FUNCTION_BLOCK FB_Fixture222 EXTENDS FB_UniversalFixture
VAR_INPUT
END_VAR
VAR_OUTPUT
END_VAR
VAR
	(*
		Add fixture sensors and actuators
	*)
END_VAR

SUPER^();

(*
	Add FB instances
*)

METHOD PROTECTED MS_Close
VAR_INPUT
END_VAR
eFixtureState := UNIVERSAL_FIXTURE_CLOSE_DONE;
END_METHOD

METHOD PROTECTED MS_Open
VAR_INPUT
END_VAR
eFixtureState := UNIVERSAL_FIXTURE_OPEN_DONE;
END_METHOD

METHOD PROTECTED MS_ReadyInitialized
VAR_INPUT
END_VAR
eFixtureState := UNIVERSAL_FIXTURE_IDLE;
END_METHOD

METHOD PROTECTED MS_Reset
VAR_INPUT
END_VAR
eFixtureState := UNIVERSAL_FIXTURE_RESET_DONE;
END_METHOD

PROPERTY SocketOpen : REFERENCE TO BOOL
GET
SocketOpen REF= bSocketOpen;
END_GET
END_PROPERTY

END_FUNCTION_BLOCK

(* stored: Version 1.1.0.1, ProductVersion 3.1.4024.9
   POU FB_Fixture222: Id {bf130327-fb73-4e0f-a2a5-8f36b7838545}, SpecialFunc None
   Method MS_Close: Id {c4fae21c-7515-4366-9c31-95e21cfd07b3}
   Method MS_Open: Id {6b0f9600-504b-4b29-844f-b9e27450c2c0}
   Method MS_ReadyInitialized: Id {669ad9b1-e38b-40bd-b030-a833d680838e}
   Method MS_Reset: Id {15b0e0ae-5769-4b30-8683-4a429256e2bc}
   Property SocketOpen: Id {91cf3a16-c367-498a-ac19-7a1da53003c2}
   Get Get: Id {e67ddd63-a741-4b80-a0bc-23a1d907c23c} *)
